TYPE Sfts_Settings_DUT :
STRUCT
	ID:  DINT;
	LP_Timeout:  UInt;
END_STRUCT
END_TYPE

(* stored: Version 1.1.0.1
   DUT Sfts_Settings_DUT: Id {d0153082-6246-41b9-a74e-d03a657fd1cc} *)
